// Mitsubishi GX Works2 project: Ex2_GROUP14   PLC: FX3G

// global labels: Global1
VAR_GLOBAL
  StartDay AT X007 : BOOL;
  StartProduction AT X001 : BOOL;
  StartCooling AT X002 : BOOL;
  Temp10Sensor AT X003 : BOOL;
  EmergencyStop AT X005 : BOOL;
  WorkingDayLight AT Y007 : BOOL;
  FlavorProcessLight AT Y000 : BOOL;
  CoolingProcessLight AT Y002 : BOOL;
  MixingLight1 AT Y005 : BOOL;
  MixingLight2 AT Y006 : BOOL;
  WorkingDay AT M0 : BOOL;
  RegularGumigum AT M15 : BOOL;
  PremiumGumigum AT M16 : BOOL;
  LackOfStock AT M20 : BOOL;
  FlavorPreparation AT M21 : BOOL;
  FlavorProcessed AT M22 : BOOL;
  SampleDone AT M19 : BOOL;
  CoolingProcessActive AT M23 : BOOL;
  CoolingProcessDone AT M24 : BOOL;
  MixingProcessActive AT M25 : BOOL;
  MixingProcessDone AT M26 : BOOL;
  EndOfDay AT M27 : BOOL;
  InitRaspberryStock AT D1100 : REAL;
  RaspberryStock AT D1112 : REAL;
  InitLemonStock AT D1114 : REAL;
  LemonStock AT D1116 : REAL;
  InitStabilizerStock AT D1118 : REAL;
  StabilizerStock AT D1120 : REAL;
  InitGummyBearsStock AT D1122 : REAL;
  GummyBearsStock AT D1124 : REAL;
  PackagesCounter AT D1126 : REAL;
  AnalogInput1 AT D8280 : INT;
  SampledAnalogInput AT D1130 : INT;
  AnalogInputFloat AT D1132 : REAL;
  AnalogOutput AT D8282 : REAL;
  OutputPackagesFloat AT D1134 : REAL;
END_VAR
VAR_GLOBAL CONSTANT
  ConstRegularGumigum : REAL := 2000;
  ConstPremiumGumigum : REAL := 4000;
  RaspberryStockConstR : REAL := 280.0;
  LemonStockConstR : REAL := 455.0;
  StabilizerStockConstR : REAL := 105.0;
  GummyBearsStockConstR : REAL := 28.0;
  RaspberryStockConstP : REAL := 385.0;
  LemonStockConstP : REAL := 665.0;
  StabilizerStockConstP : REAL := 210.0;
  GummyBearsStockConstP : REAL := 70.0;
  RaspberryIceCreamConstR : REAL := 350.0;
  LemonIceCreamConstR : REAL := 490.0;
  RaspberryIceCreamConstP : REAL := 560.0;
  LemonIceCreamConstP : REAL := 700.0;
  DivideByTen : REAL := 10.0;
END_VAR
VAR_GLOBAL
  RaspberryIceCreamContainer AT D1152 : REAL;
  LemonIceCreamContainer AT D1154 : REAL;
  RaspberryIceCreamCooling AT D1156 : REAL;
  LemonIceCreamCooling AT D1158 : REAL;
  MixingTank AT D1160 : REAL;
  FlavorTimer AT TC5 : BOOL;
  FlavorTimerDone AT TS5 : BOOL;
  CoolingTimer AT TC8 : BOOL;
  CoolingTimerDone AT TS8 : BOOL;
  MixingTimerRegular AT TC10 : BOOL;
  MixingTimerRegularDone AT TS10 : BOOL;
  MixingTimerPremium AT TC11 : BOOL;
  MixingTimerPremiumDone AT TS11 : BOOL;
  FirstBlinkTimer AT TC12 : BOOL;
  FirstBlinkTimerDone AT TS12 : BOOL;
  SecondBlinkTimer AT TC13 : BOOL;
  SecondBlinkTimerDone AT TS13 : BOOL;
  CoolingCanStart AT M33 : BOOL;
  MixingCanStart AT M34 : BOOL;
END_VAR
VAR_GLOBAL CONSTANT
  Time5Sec : INT := 50;
  Time8Sec : INT := 80;
  Time3Sec : INT := 30;
  Time05Sec : INT := 5;
  ResetFloat : REAL;
  ResetWord : INT;
  OnePackage : REAL := 1.0;
END_VAR
VAR_GLOBAL
  LackRaspR AT M40 : BOOL;
  LackLemonR AT M41 : BOOL;
  LackStabR AT M42 : BOOL;
  LackGummyR AT M43 : BOOL;
  LackRaspP AT M44 : BOOL;
  LackLemonP AT M45 : BOOL;
  LackStabP AT M46 : BOOL;
  LackGummyP AT M47 : BOOL;
  ResetAll AT M36 : BOOL;
END_VAR

// task Task_01 (event TRUE, interval 0, priority 31): POU_01

PROGRAM POU_01
(* structured ladder/FBD written out as ST: instructions are called as NAME(EN, inputs, outputs); _pN, _eN, _tN stand for wires *)
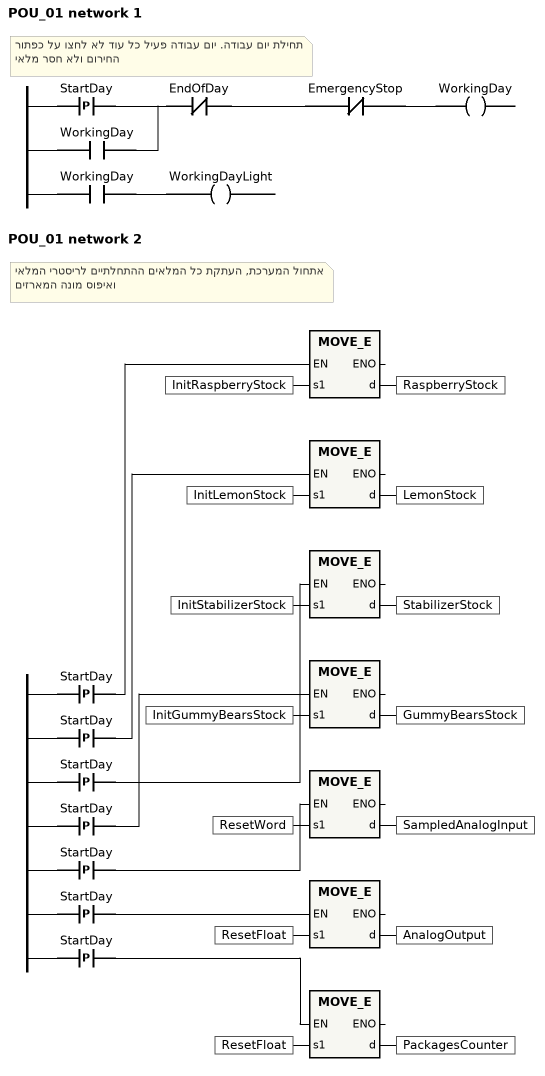
(* network 1 *)
(* תחילת יום עבודה. יום עבודה פעיל כל עוד לא לחצו על כפתור החירום ולא חסר מלאי *)
WorkingDay := ((LDP(TRUE, StartDay) OR WorkingDay) AND NOT EndOfDay) AND NOT EmergencyStop;
WorkingDayLight := WorkingDay;
(* network 2 *)
(* אתחול המערכת, העתקת כל המלאים ההתחלתיים לריסטרי המלאי ואיפוס מונה המארזים *)
MOVE_E(LDP(TRUE, StartDay), InitRaspberryStock, RaspberryStock);
MOVE_E(LDP(TRUE, StartDay), InitLemonStock, LemonStock);
MOVE_E(LDP(TRUE, StartDay), InitStabilizerStock, StabilizerStock);
MOVE_E(LDP(TRUE, StartDay), InitGummyBearsStock, GummyBearsStock);
MOVE_E(LDP(TRUE, StartDay), ResetWord, SampledAnalogInput);
MOVE_E(LDP(TRUE, StartDay), ResetFloat, AnalogOutput);
MOVE_E(LDP(TRUE, StartDay), ResetFloat, PackagesCounter);
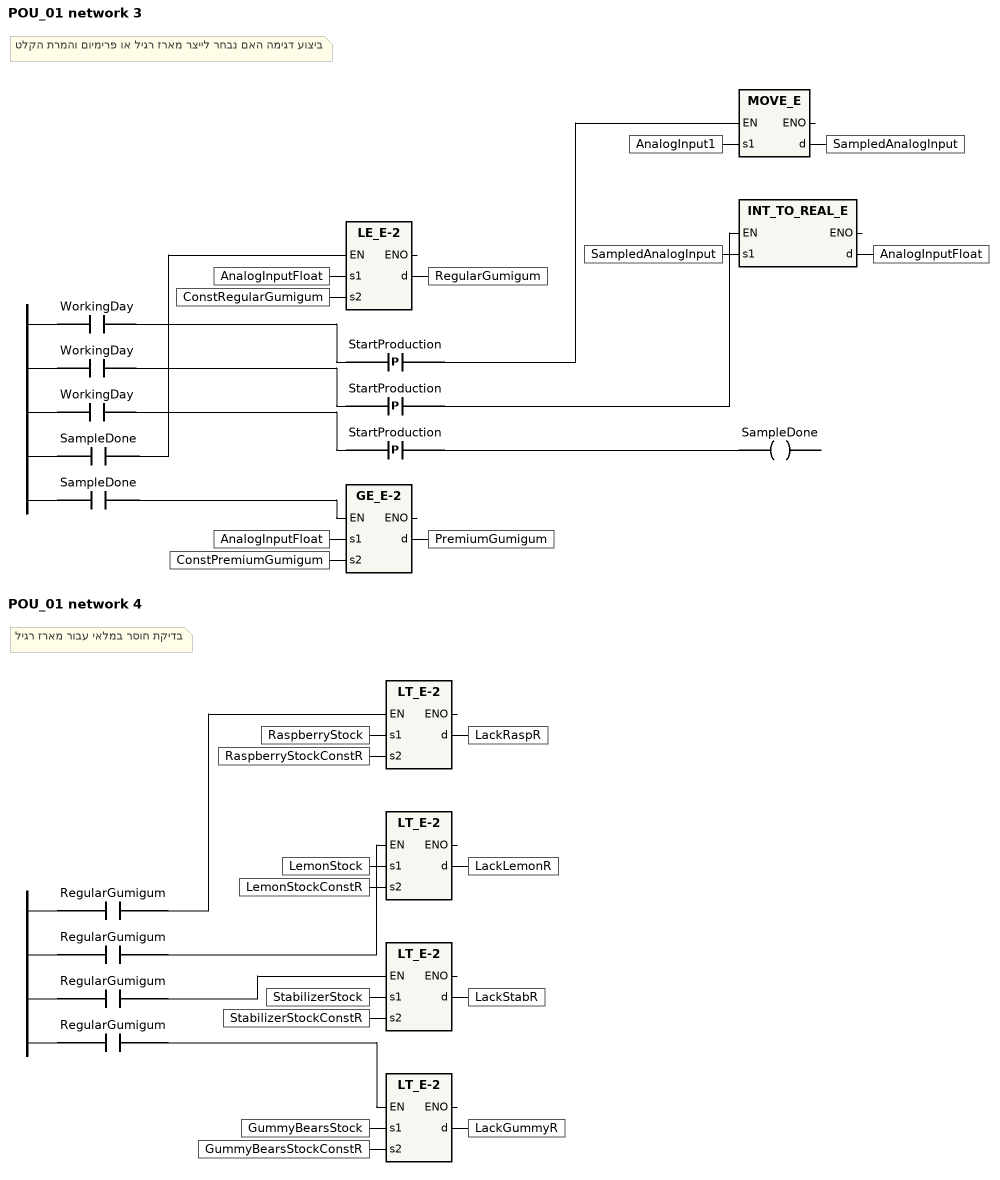
(* network 3 *)
(* ביצוע דגימה האם נבחר לייצר מארז רגיל או פרימיום והמרת הקלט *)
MOVE_E(WorkingDay AND LDP(TRUE, StartProduction), AnalogInput1, SampledAnalogInput);
INT_TO_REAL_E(WorkingDay AND LDP(TRUE, StartProduction), SampledAnalogInput, AnalogInputFloat);
SampleDone := WorkingDay AND LDP(TRUE, StartProduction);
LE_E(SampleDone, AnalogInputFloat, ConstRegularGumigum, RegularGumigum);
GE_E(SampleDone, AnalogInputFloat, ConstPremiumGumigum, PremiumGumigum);
(* network 4 *)
(* בדיקת חוסר במלאי עבור מארז רגיל *)
LT_E(RegularGumigum, RaspberryStock, RaspberryStockConstR, LackRaspR);
LT_E(RegularGumigum, LemonStock, LemonStockConstR, LackLemonR);
LT_E(RegularGumigum, StabilizerStock, StabilizerStockConstR, LackStabR);
LT_E(RegularGumigum, GummyBearsStock, GummyBearsStockConstR, LackGummyR);
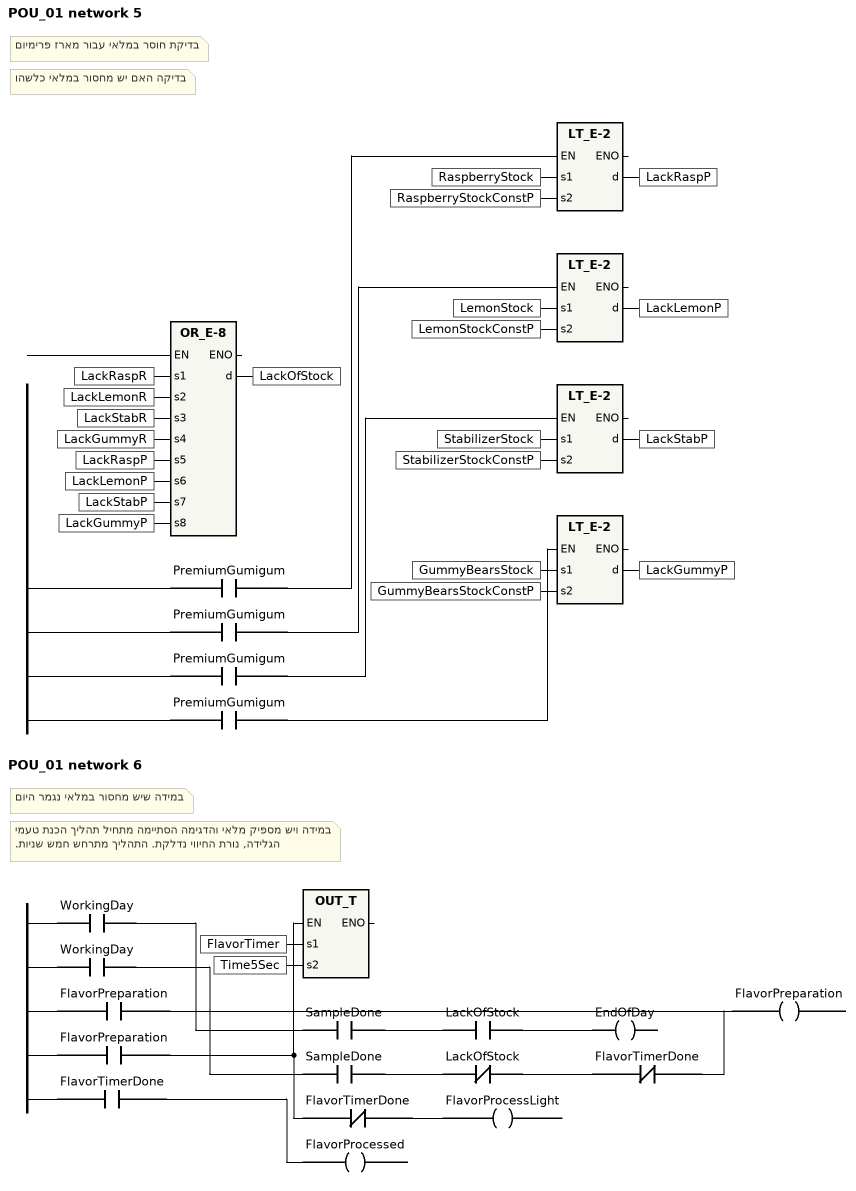
(* network 5 *)
(* בדיקת חוסר במלאי עבור מארז פרימיום *)
(* בדיקה האם יש מחסור במלאי כלשהו *)
LT_E(PremiumGumigum, RaspberryStock, RaspberryStockConstP, LackRaspP);
LT_E(PremiumGumigum, LemonStock, LemonStockConstP, LackLemonP);
LT_E(PremiumGumigum, StabilizerStock, StabilizerStockConstP, LackStabP);
LT_E(PremiumGumigum, GummyBearsStock, GummyBearsStockConstP, LackGummyP);
OR_E(TRUE, LackRaspR, LackLemonR, LackStabR, LackGummyR, LackRaspP, LackLemonP, LackStabP, LackGummyP, LackOfStock);
(* network 6 *)
(* במידה שיש מחסור במלאי נגמר היום *)
(* במידה ויש מספיק מלאי והדגימה הסתיימה מתחיל תהליך הכנת טעמי הגלידה, נורת החיווי נדלקת. התהליך מתרחש חמש שניות. *)
EndOfDay := WorkingDay AND SampleDone AND LackOfStock;
FlavorPreparation := (WorkingDay AND SampleDone AND NOT LackOfStock AND NOT FlavorTimerDone) OR FlavorPreparation;
OUT_T(FlavorPreparation, FlavorTimer, Time5Sec);
FlavorProcessLight := FlavorPreparation AND NOT FlavorTimerDone;
FlavorProcessed := FlavorTimerDone;
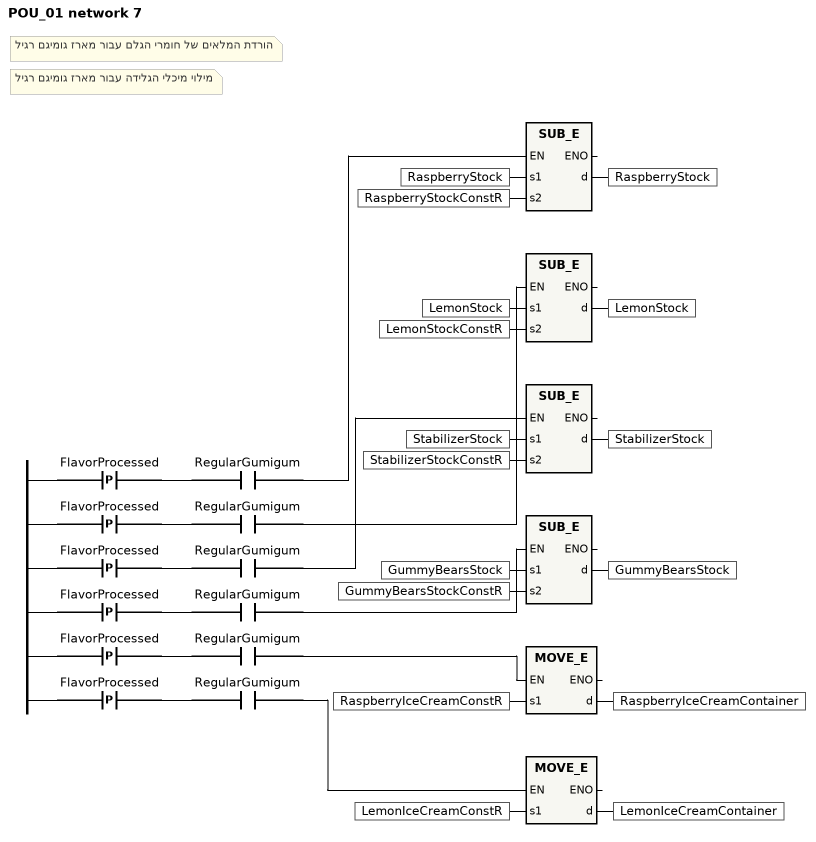
(* network 7 *)
(* הורדת המלאים של חומרי הגלם עבור מארז גומיגם רגיל *)
(* מילוי מיכלי הגלידה עבור מארז גומיגם רגיל *)
SUB_E(LDP(TRUE, FlavorProcessed) AND RegularGumigum, RaspberryStock, RaspberryStockConstR, RaspberryStock);
SUB_E(LDP(TRUE, FlavorProcessed) AND RegularGumigum, LemonStock, LemonStockConstR, LemonStock);
SUB_E(LDP(TRUE, FlavorProcessed) AND RegularGumigum, StabilizerStock, StabilizerStockConstR, StabilizerStock);
SUB_E(LDP(TRUE, FlavorProcessed) AND RegularGumigum, GummyBearsStock, GummyBearsStockConstR, GummyBearsStock);
MOVE_E(LDP(TRUE, FlavorProcessed) AND RegularGumigum, RaspberryIceCreamConstR, RaspberryIceCreamContainer);
MOVE_E(LDP(TRUE, FlavorProcessed) AND RegularGumigum, LemonIceCreamConstR, LemonIceCreamContainer);
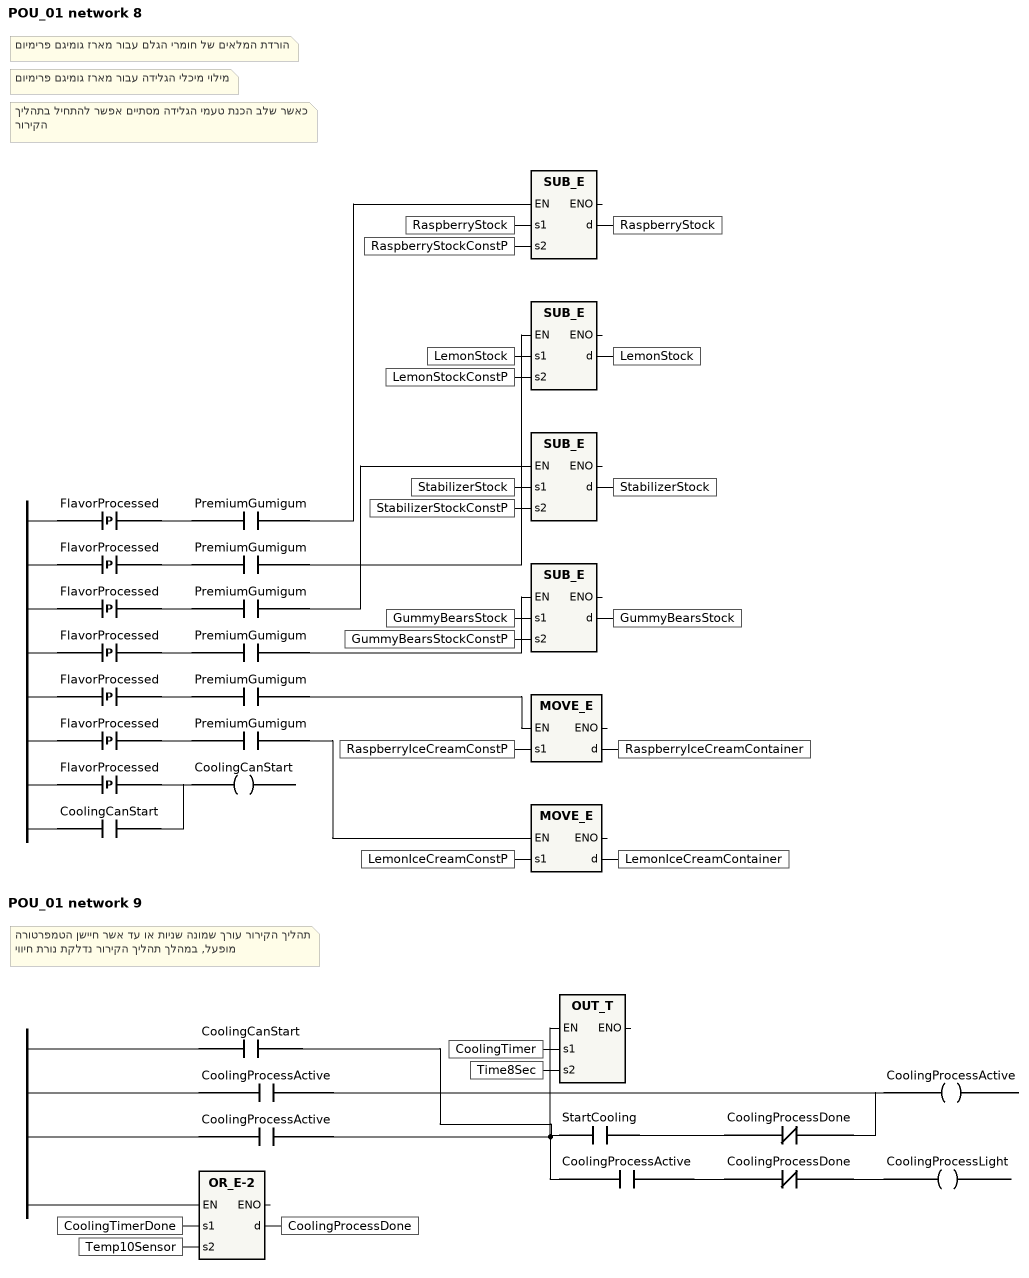
(* network 8 *)
(* הורדת המלאים של חומרי הגלם עבור מארז גומיגם פרימיום *)
(* מילוי מיכלי הגלידה עבור מארז גומיגם פרימיום *)
(* כאשר שלב הכנת טעמי הגלידה מסתיים אפשר להתחיל בתהליך הקירור *)
SUB_E(LDP(TRUE, FlavorProcessed) AND PremiumGumigum, RaspberryStock, RaspberryStockConstP, RaspberryStock);
SUB_E(LDP(TRUE, FlavorProcessed) AND PremiumGumigum, LemonStock, LemonStockConstP, LemonStock);
SUB_E(LDP(TRUE, FlavorProcessed) AND PremiumGumigum, StabilizerStock, StabilizerStockConstP, StabilizerStock);
SUB_E(LDP(TRUE, FlavorProcessed) AND PremiumGumigum, GummyBearsStock, GummyBearsStockConstP, GummyBearsStock);
MOVE_E(LDP(TRUE, FlavorProcessed) AND PremiumGumigum, RaspberryIceCreamConstP, RaspberryIceCreamContainer);
MOVE_E(LDP(TRUE, FlavorProcessed) AND PremiumGumigum, LemonIceCreamConstP, LemonIceCreamContainer);
CoolingCanStart := LDP(TRUE, FlavorProcessed) OR CoolingCanStart;
(* network 9 *)
(* תהליך הקירור עורך שמונה שניות או עד אשר חיישן הטמפרטורה מופעל, במהלך תהליך הקירור נדלקת נורת חיווי *)
CoolingProcessActive := (CoolingCanStart AND StartCooling AND NOT CoolingProcessDone) OR CoolingProcessActive;
OUT_T(CoolingProcessActive, CoolingTimer, Time8Sec);
CoolingProcessLight := CoolingProcessActive AND CoolingProcessActive AND NOT CoolingProcessDone;
OR_E(TRUE, CoolingTimerDone, Temp10Sensor, CoolingProcessDone);
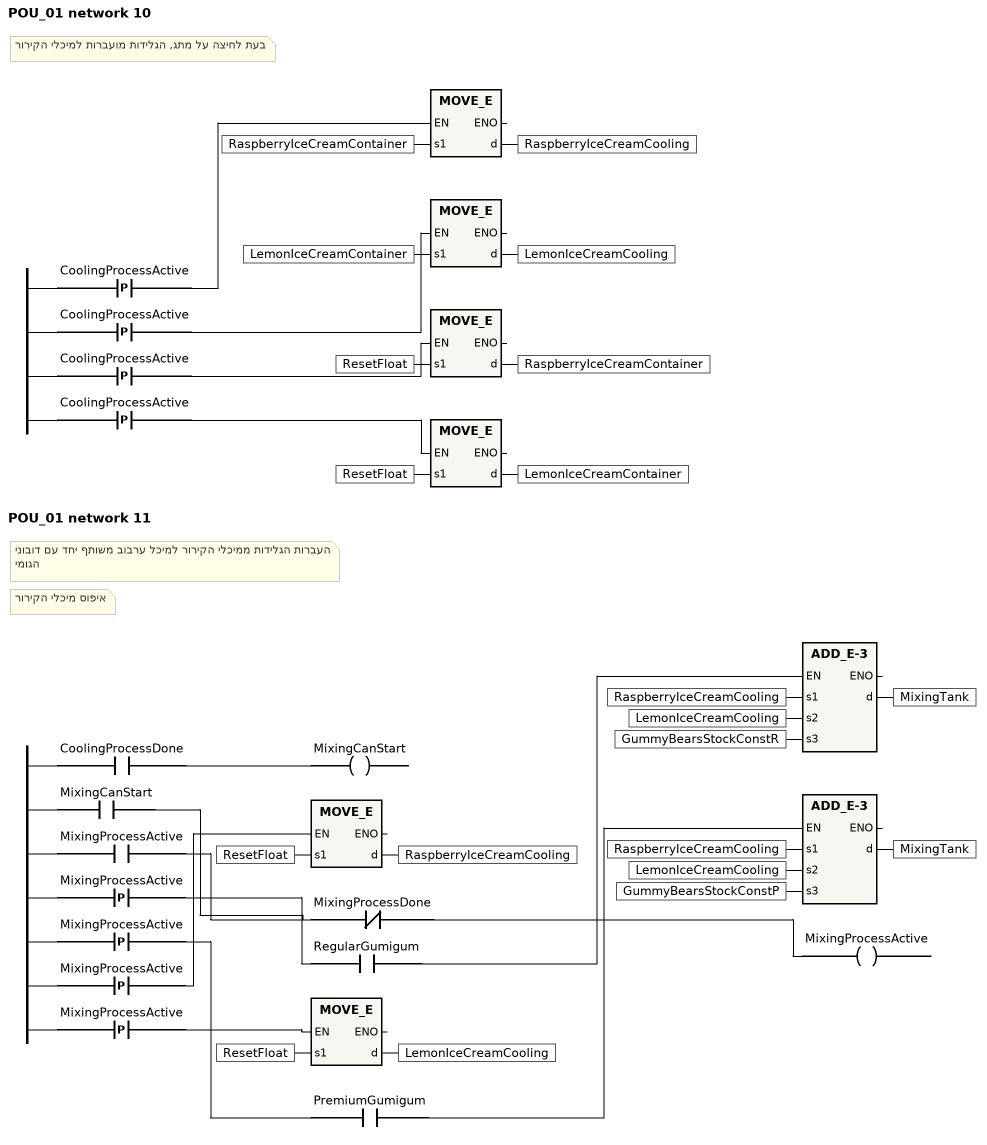
(* network 10 *)
(* בעת לחיצה על מתג, הגלידות מועברות למיכלי הקירור *)
MOVE_E(LDP(TRUE, CoolingProcessActive), RaspberryIceCreamContainer, RaspberryIceCreamCooling);
MOVE_E(LDP(TRUE, CoolingProcessActive), LemonIceCreamContainer, LemonIceCreamCooling);
MOVE_E(LDP(TRUE, CoolingProcessActive), ResetFloat, RaspberryIceCreamContainer);
MOVE_E(LDP(TRUE, CoolingProcessActive), ResetFloat, LemonIceCreamContainer);
(* network 11 *)
(* העברות הגלידות ממיכלי הקירור למיכל ערבוב משותף יחד עם דובוני הגומי *)
(* איפוס מיכלי הקירור *)
MixingCanStart := CoolingProcessDone;
MixingProcessActive := (MixingCanStart OR MixingProcessActive) AND NOT MixingProcessDone;
ADD_E(LDP(TRUE, MixingProcessActive) AND RegularGumigum, RaspberryIceCreamCooling, LemonIceCreamCooling, GummyBearsStockConstR, MixingTank);
ADD_E(LDP(TRUE, MixingProcessActive) AND PremiumGumigum, RaspberryIceCreamCooling, LemonIceCreamCooling, GummyBearsStockConstP, MixingTank);
MOVE_E(LDP(TRUE, MixingProcessActive), ResetFloat, RaspberryIceCreamCooling);
MOVE_E(LDP(TRUE, MixingProcessActive), ResetFloat, LemonIceCreamCooling);
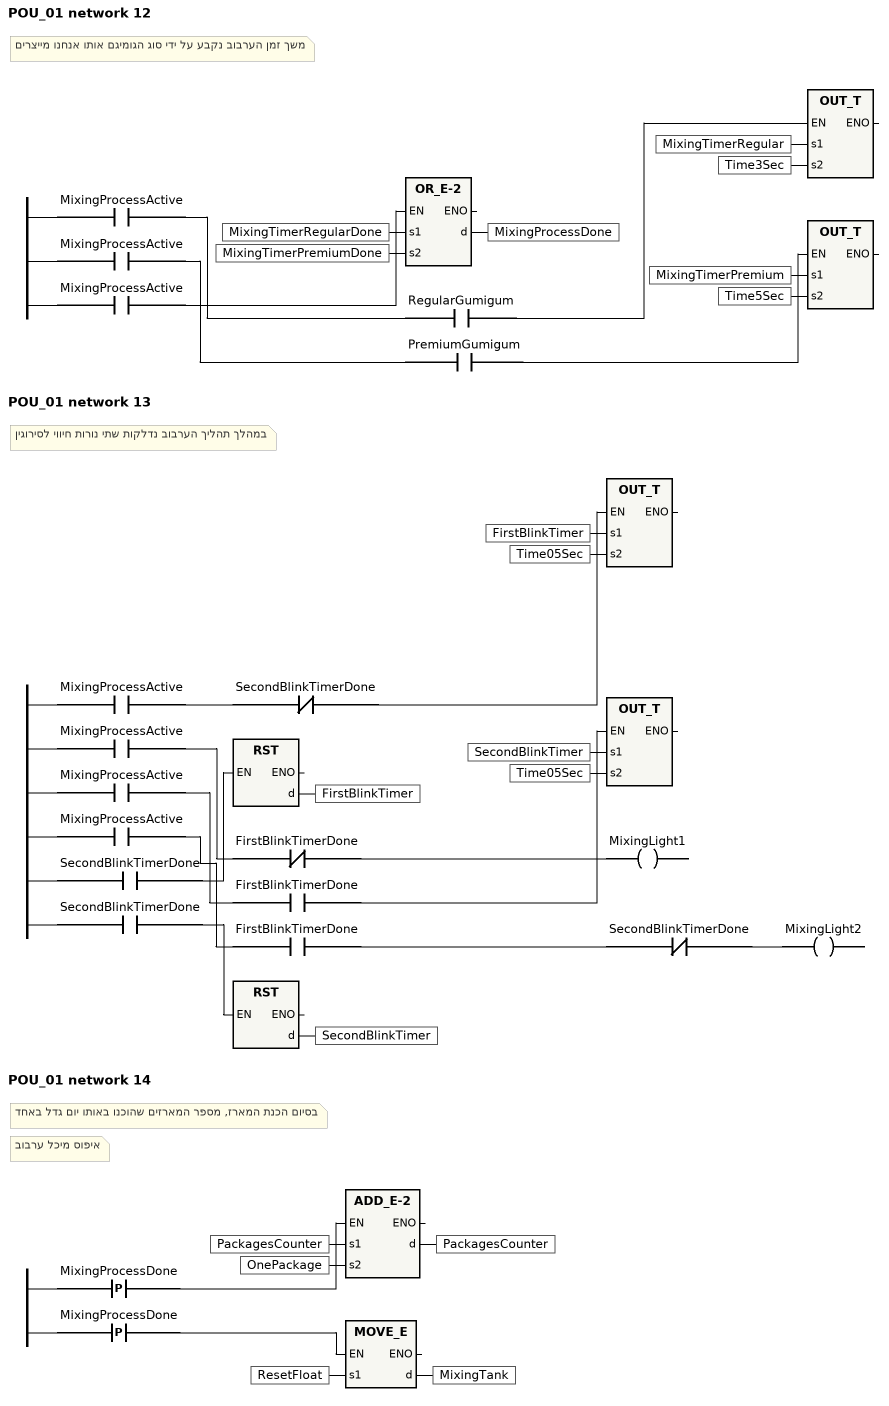
(* network 12 *)
(* משך זמן הערבוב נקבע על ידי סוג הגומיגם אותו אנחנו מייצרים *)
OUT_T(MixingProcessActive AND RegularGumigum, MixingTimerRegular, Time3Sec);
OUT_T(MixingProcessActive AND PremiumGumigum, MixingTimerPremium, Time5Sec);
OR_E(MixingProcessActive, MixingTimerRegularDone, MixingTimerPremiumDone, MixingProcessDone);
(* network 13 *)
(* במהלך תהליך הערבוב נדלקות שתי נורות חיווי לסירוגין *)
OUT_T(MixingProcessActive AND NOT SecondBlinkTimerDone, FirstBlinkTimer, Time05Sec);
MixingLight1 := MixingProcessActive AND NOT FirstBlinkTimerDone;
OUT_T(MixingProcessActive AND FirstBlinkTimerDone, SecondBlinkTimer, Time05Sec);
MixingLight2 := MixingProcessActive AND FirstBlinkTimerDone AND NOT SecondBlinkTimerDone;
RST(SecondBlinkTimerDone, FirstBlinkTimer);
RST(SecondBlinkTimerDone, SecondBlinkTimer);
(* network 14 *)
(* בסיום הכנת המארז, מספר המארזים שהוכנו באותו יום גדל באחד *)
(* איפוס מיכל ערבוב *)
ADD_E(LDP(TRUE, MixingProcessDone), PackagesCounter, OnePackage, PackagesCounter);
MOVE_E(LDP(TRUE, MixingProcessDone), ResetFloat, MixingTank);
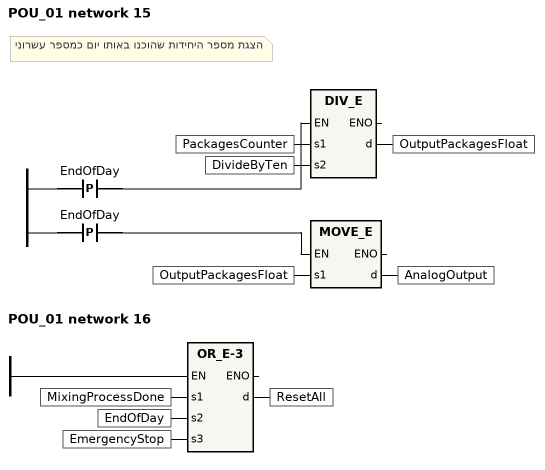
(* network 15 *)
(* הצגת מספר היחידות שהוכנו באותו יום כמספר עשרוני *)
DIV_E(LDP(TRUE, EndOfDay), PackagesCounter, DivideByTen, OutputPackagesFloat);
MOVE_E(LDP(TRUE, EndOfDay), OutputPackagesFloat, AnalogOutput);
(* network 16 *)
OR_E(TRUE, MixingProcessDone, EndOfDay, EmergencyStop, ResetAll);
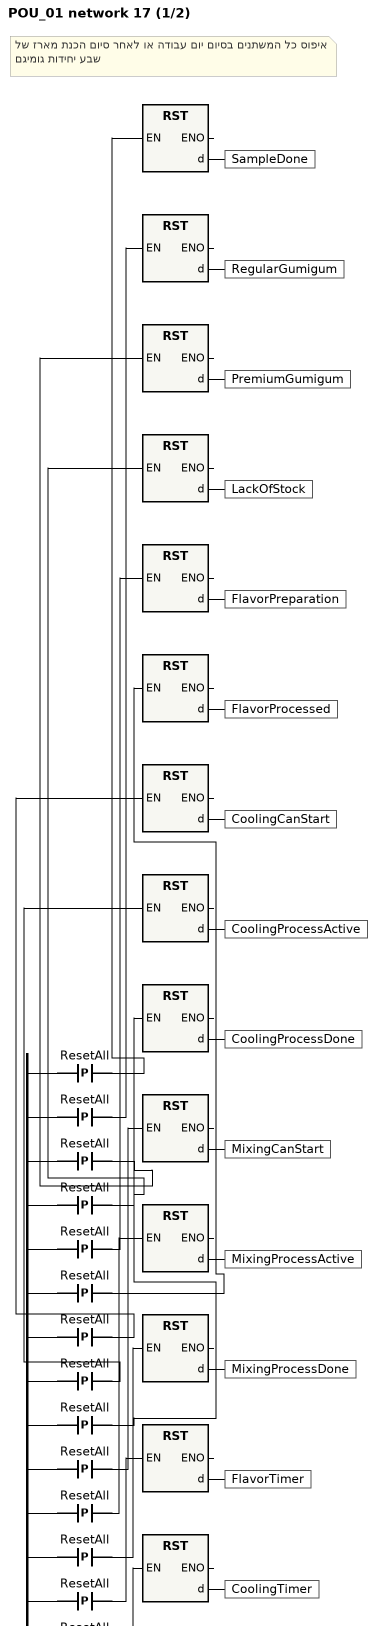
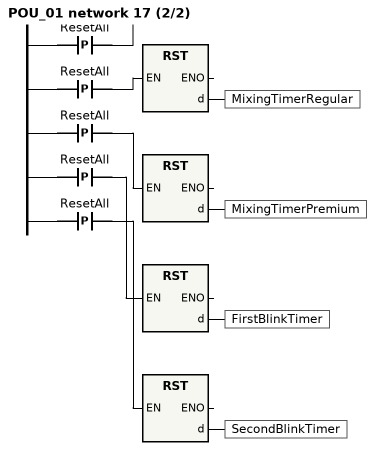
(* network 17 *)
(* איפוס כל המשתנים בסיום יום עבודה או לאחר סיום הכנת מארז של שבע יחידות גומיגם *)
RST(LDP(TRUE, ResetAll), SampleDone);
RST(LDP(TRUE, ResetAll), RegularGumigum);
RST(LDP(TRUE, ResetAll), PremiumGumigum);
RST(LDP(TRUE, ResetAll), LackOfStock);
RST(LDP(TRUE, ResetAll), FlavorPreparation);
RST(LDP(TRUE, ResetAll), FlavorProcessed);
RST(LDP(TRUE, ResetAll), CoolingCanStart);
RST(LDP(TRUE, ResetAll), CoolingProcessActive);
RST(LDP(TRUE, ResetAll), CoolingProcessDone);
RST(LDP(TRUE, ResetAll), MixingCanStart);
RST(LDP(TRUE, ResetAll), MixingProcessActive);
RST(LDP(TRUE, ResetAll), MixingProcessDone);
RST(LDP(TRUE, ResetAll), FlavorTimer);
RST(LDP(TRUE, ResetAll), CoolingTimer);
RST(LDP(TRUE, ResetAll), MixingTimerRegular);
RST(LDP(TRUE, ResetAll), MixingTimerPremium);
RST(LDP(TRUE, ResetAll), FirstBlinkTimer);
RST(LDP(TRUE, ResetAll), SecondBlinkTimer);
END_PROGRAM
